PROGRAM ReadModbusReg
VAR
	fbReadRegs        : FB_MBReadRegs;
    bReadRegs         : BOOL;
    bReadRegsBusy     : BOOL;
    bReadRegsError    : BOOL;
    nReadRegsErrorId  : UDINT;
    nReadRegsCount    : UDINT;
    nQuantity         : WORD:=2;
    nMBAddr           : WORD:=32768;
    arrData           : ARRAY [0..1] OF WORD;
	nTCPPort		  : UINT	:= 502;
	nUnitID			  : BYTE	:= 255;
	tTimeout		  : TIME	:= T#1S;
END_VAR

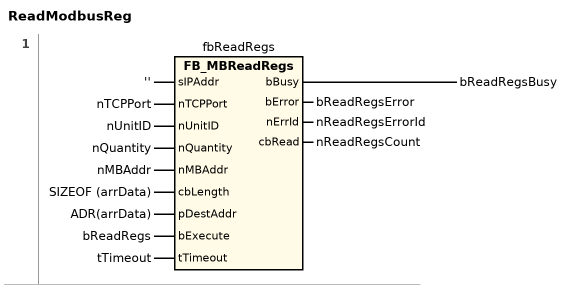
// NETWORK 1
fbReadRegs(
    sIPAddr := '',
    nTCPPort := nTCPPort,
    nUnitID := nUnitID,
    nQuantity := nQuantity,
    nMBAddr := nMBAddr,
    cbLength := SIZEOF (arrData),
    pDestAddr := ADR(arrData),
    bExecute := bReadRegs,
    tTimeout := tTimeout,
    bError => bReadRegsError,
    nErrId => nReadRegsErrorId,
    cbRead => nReadRegsCount); // FB_MBReadRegs
bReadRegsBusy := fbReadRegs.bBusy;

END_PROGRAM

(* stored: Version 1.1.0.1, ProductVersion 3.1.4024.12
   POU ReadModbusReg: Id {6dc804f7-b739-4af5-bbb9-2b41f9b25d30}, SpecialFunc None *)
